// This function has been automatically generated from the project information.
{attribute 'signature_flag' := '1073741824'}
{attribute 'TcGenerated'}
{attribute 'no-analysis'}
FUNCTION F_GetTitle : WSTRING
VAR_INPUT
	
END_VAR

F_GetTitle := "RoofTrussLibrary";

END_FUNCTION

(* stored: Version 1.1.0.1
   POU F_GetTitle: Id {2d56814f-f70f-4003-a27d-e963246a8842}, SpecialFunc None *)
